FUNCTION_BLOCK CONTROL_SPIRAL_MOVE
  (* Standard: 61499-2 *)
  (* Version 1.0, 31/05/2012, GASR *)
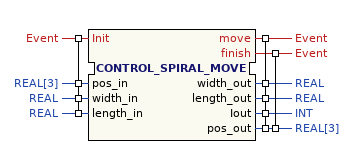
  EVENT_INPUT
    Init WITH width_in, length_in, pos_in; (* first time execution *)
  END_EVENT
  EVENT_OUTPUT
    move WITH width_out, length_out, pos_out, Iout;
    finish WITH pos_out;
  END_EVENT
  VAR_INPUT
    pos_in : ARRAY [0..2] OF REAL;
    width_in : REAL;
    length_in : REAL;
  END_VAR
  VAR_OUTPUT
    width_out : REAL;
    length_out : REAL;
    Iout : INT := 0;
    pos_out : ARRAY [0..2] OF REAL;
  END_VAR
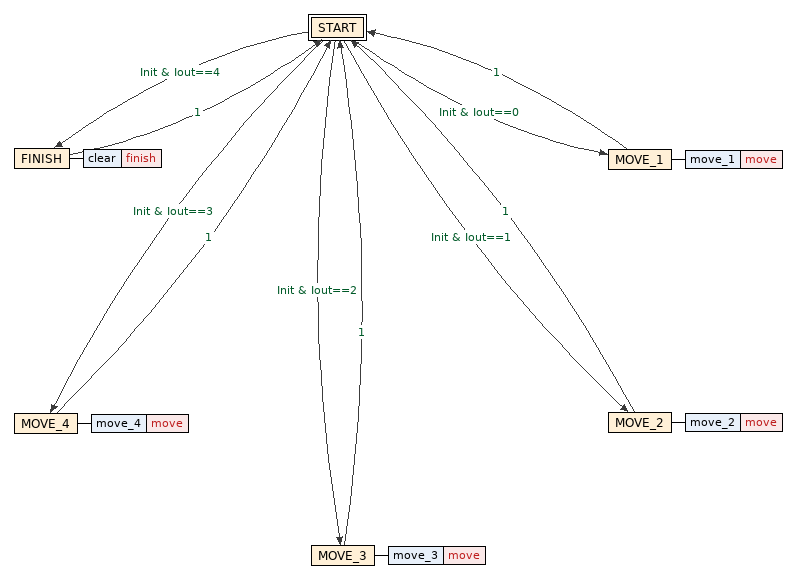
  EC_STATES
    START;
    MOVE_1 : move_1 -> move;
    MOVE_2 : move_2 -> move;
    MOVE_3 : move_3 -> move;
    MOVE_4 : move_4 -> move;
    FINISH : clear -> finish;
  END_STATES
  EC_TRANSITIONS
    START TO MOVE_1 := Init & Iout==0;
    START TO MOVE_2 := Init & Iout==1;
    START TO MOVE_3 := Init & Iout==2;
    START TO MOVE_4 := Init & Iout==3;
    START TO FINISH := Init & Iout==4;
    MOVE_1 TO START := 1;
    MOVE_2 TO START := 1;
    MOVE_3 TO START := 1;
    MOVE_4 TO START := 1;
    FINISH TO START := 1;
  END_TRANSITIONS
  ALGORITHM move_1 IN Lua:
			length_out = length_in
			width_out = 0
			Iout = Iout + 1
			pos_out = {pos_in[1], pos_in[2], pos_in[3]}
  END_ALGORITHM
  ALGORITHM move_2 IN Lua:
			length_out = 0
			width_out = width_in
			Iout = Iout + 1
			pos_out = {pos_in[1], pos_in[2], pos_in[3]}
  END_ALGORITHM
  ALGORITHM move_3 IN Lua:
			length_out = -length_in
			width_out = 0
			Iout = Iout + 1
			pos_out = {pos_in[1], pos_in[2], pos_in[3]}
  END_ALGORITHM
  ALGORITHM move_4 IN Lua:
			length_out = 0
			width_out = -width_in
			Iout = Iout + 1
			pos_out = {pos_in[1], pos_in[2], pos_in[3]}
  END_ALGORITHM
  ALGORITHM clear IN Lua:
			Iout = 0
			pos_out = pos_in
  END_ALGORITHM
END_FUNCTION_BLOCK
